// TIA Portal V20 export
VAR_GLOBAL   // PLC tag table "LGR_Const_Gripper"
END_VAR
VAR_GLOBAL CONSTANT   // user constants
   GRIP_IDLE : USInt := 0;   // no request / 요청 없음
   GRIP_MOVE : USInt := 1;   // move without torque change / 토크 변경 없이 이동
   GRIP_GRIP : USInt := 2;   // open grip / OPEN 파지 (벌림)
   GRIP_CLOSE : USInt := 3;   // close (pre-grip / release) / CLOSE 오므림 (프리그립 / 해제)
   GRIP_MEASURE_OPEN : USInt := 4;   // measure open (contact detect) / 측정 저힘 벌림 (접촉 판정)
   GRIP_RETRY : USInt := 5;   // retry grip / 재파지 벌림
   GRIP_LEARN : USInt := 6;   // learn mechanism load (no tire) / 기구 부하 학습 (타이어 없이)
   GRIP_LIMIT : USInt := 7;   // set torque limit only (no move) / 토크 제한만 설정 (이동 없음, 재시도 Z 하강)
   GRIP_OWNER_TASK : USInt := 1;   // PL_Task_V2
   GRIP_OWNER_MEASURE : USInt := 2;   // PL_MeasureItem
   GRIP_OWNER_MANUAL_MEASURE : USInt := 3;   // PL_ManualMeasureItem
   GRIP_OWNER_MANUAL : USInt := 4;   // PL_ManualCommand
   GRIP_OWNER_LEARN : USInt := 5;   // LEARN (HMI / console)
   GRIP_ST_IDLE : USInt := 0;   // idle / 정지, 그 외
   GRIP_ST_RELEASED : USInt := 10;   // released / 정지, 화물 없음, 해제 위치
   GRIP_ST_OPENING : USInt := 20;   // opening / OPEN 방향 이동 중
   GRIP_ST_CLOSING : USInt := 30;   // closing / CLOSE 방향 이동 중
   GRIP_ST_GRIPPED_EMPTY : USInt := 40;   // torque stop without item / 토크 정지, 화물 없음 (헛파지)
   GRIP_ST_HOLDING : USInt := 50;   // holding item / 파지 유지
   GRIP_ST_MEASURING : USInt := 60;   // measuring / 측정 벌림 진행 중
   GRIP_ST_LEARNING : USInt := 65;   // learning / 기구 부하 학습 중
   GRIP_ST_STALLED : USInt := 70;   // stalled without torque / 토크 없이 정지 (안 움직임)
   GRIP_ST_TIMEOUT : USInt := 80;   // timeout / 판정 타임아웃
   GRIP_ST_OBSTACLE : USInt := 90;   // obstacle / 걸림 (삐뚤어짐)
   GRIP_ST_THERMAL : USInt := 92;   // thermal protection / 과열 보호
   GRIP_ST_FAULT : USInt := 95;   // fault / 드라이브 Fault / 요청 에러
   GRIP_E_NONE : USInt := 0;
   GRIP_E_BUSY : USInt := 1;   // busy with another owner / 다른 Owner 요청 진행 중
   GRIP_E_TORQ_ECHO : USInt := 2;   // torque limit not applied / 토크 제한 반영 안 됨
   GRIP_E_RANGE_MAX : USInt := 3;   // reached RangeMax without contact / 접촉 없이 RangeMax
   GRIP_E_ABORT : USInt := 4;   // aborted / 요청 중단
   GRIP_E_TIMEOUT : USInt := 5;   // timeout / 판정 타임아웃
   GRIP_E_RETRY_EXHAUSTED : USInt := 6;   // retries exhausted / 내부 재파지 소진
   GRIP_E_OBSTACLE : USInt := 7;   // obstacle / 걸림
   GRIP_E_LEARN : USInt := 8;   // learn failed / 학습 실패 (곡선 / 보호 상한)
   GRIP_E_THERMAL : USInt := 9;   // thermal / 과열 보호
   GRIP_E_NOT_READY : USInt := 10;   // not ready / 홈 / Fault / 과열 로 요청 거부
   GRIP_TO_NONE : USInt := 0;
   GRIP_TO_STALL_OUT : USInt := 1;   // stall outside window / 창 밖 스톨 (4025)
   GRIP_TO_NO_ITEM : USInt := 2;   // stopped in window, no item / 창 안 정지, 화물 없음 (6016)
   GRIP_TO_GRIPPER : USInt := 3;   // gripper timeout / 그리퍼 타임아웃 (6015)
   GRIP_RS_WAIT : USInt := 0;   // Request FC result : not sent yet (busy) or result belongs to another owner / 요청 함수 결과 : 보내지 못함 (다른 요청 진행 중) 또는 다른 요청자의 결과
   GRIP_RS_BUSY : USInt := 1;   // Request FC result : sent / in progress / 요청 함수 결과 : 보냄 / 진행 중
   GRIP_RS_DONE : USInt := 2;   // Request FC result : done / 요청 함수 결과 : 완료
   GRIP_RS_ERROR : USInt := 3;   // Request FC result : error or rejected (CL_Gripper.Result.ErrorCode / Reject) / 요청 함수 결과 : 에러 또는 거부 (CL_Gripper.Result.ErrorCode / Reject)
END_VAR
